// TIA Portal V19 export
DATA_BLOCK "Setpoints_Hamba"   // DB112
{ S7_Optimized_Access := 'TRUE' }
VERSION : 0.0
// stored: AutoNumber false, MemoryReserve 0
   VAR RETAIN
      Y0904FlushTime : Int := 120;   // Valve open x sec in each CIP stage
      TT0951StartSterileTime : Real := 125.0;   // Start sterile time TT 09.51
      TT0951BarrierTemp : Real := 110.0;   // Barrier temperature TT 09.51
      TT0951BarrierTime : S5Time := S5T#15S;   // Barrier time TT 09.51
      DrainingHambaTime : S5Time := S5T#5M;   // Draining Hamba line time
      TT0950BarrierTempHigh : Real := 125.0;   // Barrier temperature TT 09.50 High
      TT0950BarrierTempLow : Real := 110.0;   // Barrier temperature TT 09.50 Low
      TT0950BarrierTimeHigh : S5Time := S5T#15S;   // Barrier time TT 09.50 High
      TT0950BarrierTimeLow : S5Time := S5T#15S;   // Barrier time TT 09.50 Low
      Y0912PurgeBarrierTime : S5Time := S5T#30S;   // Purge Product from barriet to drain
   END_VAR
BEGIN
END_DATA_BLOCK
